// TwinCAT 3 PLC project RoboConnect
// Title: RoboConnect
// Company: RoboConnect
// Author: RoboConnect_Maintainers
// ProjectVersion: 0.1.0.1
// Description: 0.1.0.0 - Update branding 0.0.25.X Adds free taks methods 0.0.24.X Addes Manufacturer & Model to TcRobot 0.0.23.x WIP Changes pos to CartesianPos, adds GetJointPositions method 0.0.22.x WIP - adds Mode prop to interface and E_RobotModeStatus 0.0.21.0 removes task from connect 0.0.20.x modifies to newr jog approach. 0.0.19.x WIP 0.0.19.0 renames Param as causes issues in dependant libs 0.0.18.0 modifies connection and taskpool 0.0.0.17 fixes queue clear method 0.0.0.16 Updates array sizes, tcp connection and other bits 0.0.0.12 changes to TCP_Recv 0.0.0.11 adds command result tasks 0.0.010 minor change to results. 0.0.0.9 added result for tasks 0.0.0.9 added timeout for tasks 0.0.0.8 added TCP receive 0.0.0.7 removes mobject queue 0.0.0.6 adds I_CommandInvoker 0.0.0.5 I_Task extends queryable 0.0.0.4 adds logging 0.0.0.3
// ProgramVersion: 3.1.4024.0
// libraries:
//   Intecre.Utilities, * (Intecre Ltd)
//   Tc2_Standard, * (Beckhoff Automation GmbH)
//   Tc2_System, * (Beckhoff Automation GmbH)
//   Tc2_TcpIp, * (Beckhoff Automation GmbH)
// project tree:
//   CommandPattern/CommandInvoker/ I_CommandInvoker.TcIO, T_CommandInvoker.TcPOU
//   CommandPattern/CommandQueue/ E_CommandPriority.TcDUT, I_CommandQueue.TcIO, T_CommandQueue.TcPOU
//   Connection/ I_Connection.TcIO, RecvBuffer.TcDUT, T_ConnectionTCPIP.TcPOU
//   Connection/Tools/ T_TcpClientConnection.TcPOU, T_TcpRecieve.TcPOU, T_TcpSend.TcPOU
//   Helpers/ F_IsAtPositionCartesian.TcPOU, F_IsAtPositionJoint.TcPOU
//   Structs and Enums/Enum/ E_BufferMode.TcDUT, E_JogType.TcDUT
//   Structs and Enums/Struct/ ST_CartesianPoint.TcDUT, ST_Dynamics.TcDUT
//   / I_RoboConnect.TcIO, RoboConnectParams.TcGVL
//   Task/ T_BoolCommandTask_1.TcPOU (excluded from build), T_CommandTask_1.TcPOU (excluded from build), T_NumberCommandTask_1.TcPOU (excluded from build), I_CommandTask.TcIO, I_Task.TcIO, I_TaskPool.TcIO, T_TaskQueue.TcPOU
//   Project Information/ F_GetCompany.TcPOU, F_GetTitle.TcPOU, F_GetVersion.TcPOU
//   Task/ResultTasks/ I_BoolResultTask.TcIO, I_NumberResultTask.TcIO
//   Version/ Global_Version.TcGVL
// real-time tasks:
//   TASK PlcTask: cycle T#10ms, priority 22, ADS port 350
//   TASK PlcTask1: cycle T#10ms, priority 21, ADS port 351

// ---- CommandPattern/CommandQueue/E_CommandPriority.TcDUT
{attribute 'qualified_only'}
{attribute 'strict'}
{attribute 'to_string'}
TYPE E_CommandPriority :
(
	LOW := 0,
  NORMAL,
  HIGH
);
END_TYPE

// ---- Connection/RecvBuffer.TcDUT
TYPE RecvBuffer : ARRAY[1..RoboConnectParams.receiveBufferSize] OF BYTE; END_TYPE

// ---- Structs and Enums/Enum/E_BufferMode.TcDUT
{attribute 'qualified_only'}
{attribute 'strict'}
TYPE
E_BufferMode :
(
  Aborting := 0,
  Buffered := 1,
  BlendingJoint := 6,
  BlendingCartesian := 7
);
END_TYPE

// ---- Structs and Enums/Enum/E_JogType.TcDUT
{attribute 'qualified_only'}
{attribute 'strict'}
TYPE E_JogType :
(
	Joint,
  Cartesian
);
END_TYPE

// ---- Structs and Enums/Struct/ST_CartesianPoint.TcDUT
TYPE ST_CartesianPoint :
STRUCT
  x : LREAL;
  y : LREAL;
  z : LREAL;
  a : LREAL;
  b : LREAL;
  c : LREAL;
END_STRUCT
END_TYPE

// ---- Structs and Enums/Struct/ST_Dynamics.TcDUT
TYPE ST_Dynamics :
STRUCT
  Velocity : LREAL;
  Accleration : LREAL;
  Deceleration : LREAL;
END_STRUCT
END_TYPE

// ---- RoboConnectParams.TcGVL
VAR_GLOBAL CONSTANT
	receiveBufferSize : UINT := 2048;
	TimeOut : TIME := T#25S;
	MAX_TASK_SIZE : UINT := 20;
END_VAR

// ---- Version/Global_Version.TcGVL
{attribute 'TcGenerated'}
{attribute 'no-analysis'}
{attribute 'linkalways'}
// This function has been automatically generated from the project information.
VAR_GLOBAL CONSTANT
	{attribute 'const_non_replaced'}
	stLibVersion_RoboConnect : ST_LibVersion := (iMajor := 0, iMinor := 1, iBuild := 0, iRevision := 1, nFlags := 0, sVersion := '0.1.0.1');
END_VAR

// ---- CommandPattern/CommandInvoker/I_CommandInvoker.TcIO
INTERFACE I_CommandInvoker

METHOD PUBLIC CyclicLogic
END_METHOD

METHOD PUBLIC Initialise : BOOL
VAR_INPUT
  commandQueue : I_CommandQueue;
END_VAR
END_METHOD

METHOD PUBLIC Reset
END_METHOD

END_INTERFACE

// ---- CommandPattern/CommandQueue/I_CommandQueue.TcIO
INTERFACE I_CommandQueue

METHOD AddHighPriority : BOOL
VAR_INPUT
  cmd : I_Task; 
END_VAR
END_METHOD

METHOD AddLowPriority : BOOL
VAR_INPUT
  cmd : I_Task; 
END_VAR
END_METHOD

METHOD AddNormalPriority : BOOL
VAR_INPUT
  cmd : I_Task; 
END_VAR
END_METHOD

METHOD Clear
END_METHOD

PROPERTY Count : UINT
GET
END_GET
END_PROPERTY

METHOD GetNext : BOOL;
VAR_OUTPUT
	output_command : I_Task;
END_VAR
END_METHOD

END_INTERFACE

// ---- Connection/I_Connection.TcIO
INTERFACE I_Connection

METHOD Connect 
VAR_INPUT
  ip : T_IPv4Addr;
  port : UINT;
  timeout : TIME;
END_VAR
END_METHOD

METHOD Disconnect
END_METHOD

PROPERTY ErrID : UDINT
GET
END_GET
END_PROPERTY

METHOD ErrorReceive : BOOL
VAR_INPUT
END_VAR
END_METHOD

PROPERTY IsBusy : BOOL
GET
END_GET
END_PROPERTY

PROPERTY IsConnected : BOOL
GET
END_GET
END_PROPERTY

PROPERTY IsErrorConnect : Bool
GET
END_GET
END_PROPERTY

PROPERTY IsErrorReceive : Bool
GET
END_GET
END_PROPERTY

PROPERTY IsErrorSend : Bool
GET
END_GET
END_PROPERTY

METHOD Receive : BOOL // TRUE if new data recieved.
VAR_OUTPUT 
  data : ARRAY [1..RoboConnectParams.receiveBufferSize] OF BYTE;  // Contents of received buffer
  receiveLength : UDINT; // length of data received.
END_VAR
END_METHOD

METHOD Send : BOOL
VAR_INPUT
  message : T_Maxstring;
END_VAR
END_METHOD

PROPERTY PUBLIC SendDone : BOOL
GET
END_GET
END_PROPERTY

END_INTERFACE

// ---- I_RoboConnect.TcIO
INTERFACE I_RoboConnect

PROPERTY CartesianPosition : ST_CartesianPoint
GET
END_GET
END_PROPERTY

METHOD ClearError : BOOL
VAR_OUTPUT
  task : I_Task;
END_VAR
END_METHOD

METHOD Connect : BOOL
//VAR_OUTPUT
//  task : I_Task;
//END_VAR
END_METHOD

PROPERTY Connected : BOOL
GET
END_GET
END_PROPERTY

METHOD CyclicLogic
END_METHOD

METHOD Disable : BOOL
VAR_OUTPUT
  task : I_Task;
END_VAR
END_METHOD

METHOD Disconnect : BOOL
VAR_OUTPUT
  task : I_Task;
END_VAR
END_METHOD

METHOD Enable : BOOL
VAR_OUTPUT
  task : I_Task;
END_VAR
END_METHOD

PROPERTY Enabled : BOOL
GET
END_GET
END_PROPERTY

PROPERTY Error : BOOL
GET
END_GET
END_PROPERTY

PROPERTY ErrorID : LREAL
GET
END_GET
END_PROPERTY

METHOD FreeAllTasks
END_METHOD

METHOD GetAnalogOutput : BOOL
VAR_INPUT
  Index : UINT;
END_VAR
VAR_OUTPUT
  task : I_NumberResultTask;
END_VAR
END_METHOD

METHOD GetAxisCurrents : BOOL
VAR_IN_OUT
  Values : ARRAY[*] OF LREAL;
END_VAR
VAR_OUTPUT
  task : I_Task;
END_VAR
END_METHOD

METHOD GetAxisPositions : BOOL
VAR_IN_OUT
  Values : ARRAY[*] OF LREAL;
END_VAR
VAR_OUTPUT
  task : I_Task;
END_VAR
END_METHOD

METHOD GetAxisTemperatures : BOOL
VAR_IN_OUT
  Values : ARRAY[*] OF LREAL;
END_VAR
VAR_OUTPUT
  task : I_Task;
END_VAR
END_METHOD

METHOD GetDigitalOutput : BOOL
VAR_INPUT
    Index : UINT;
END_VAR
VAR_OUTPUT
  task : I_BoolResultTask;
  value 	: BOOL;
END_VAR
END_METHOD

METHOD GetJointPositions : BOOL // false if incompatible array length
VAR_IN_OUT
  joints : ARRAY[*] OF LREAL; // values overwritten with joint positions.
END_VAR
END_METHOD

METHOD GetToolAnalogOutput : BOOL
VAR_INPUT
  Index : UINT;
END_VAR
VAR_OUTPUT
  task : I_NumberResultTask;
END_VAR
END_METHOD

METHOD GetToolDigitalOutput : BOOL
VAR_INPUT
  Index : UINT;
END_VAR
VAR_OUTPUT
  task : I_BoolResultTask;
END_VAR
END_METHOD

METHOD Halt : BOOL
VAR_OUTPUT
  task : I_Task;
END_VAR
END_METHOD

METHOD IsAtCartesianPosition : BOOL
VAR_INPUT
	point	: ST_CartesianPoint;
END_VAR
END_METHOD

METHOD IsAtJointPosition : BOOL
VAR_IN_OUT
  joints : ARRAY[*] OF LREAL; // positions 1..NumberOfAxes will be used. passed array should be dimensioned accordingly
END_VAR
END_METHOD

METHOD JogAxis : BOOL // default tool and user frame
VAR_INPUT
  axisIndex : UDINT; // joint or enumerated cartesian direction/vector. See concrete type docs for enumeration of cartesian coords.
  axisDirection : BOOL; // TRUE = positive, FALSE = negative
  jogType : E_JogType; // Cartesian or Joint space
END_VAR
VAR_OUTPUT
  task : I_Task;
END_VAR
END_METHOD

METHOD JogAxisAdvanced : BOOL
VAR_INPUT
  axisIndex : UDINT; // joint or enumerated cartesian direction/vector. See concrete type docs for enumeration of cartesian coords.
  axisDirection : BOOL; // TRUE = positive, FALSE = negative
  jogType : E_JogType; // Cartesian or Joint space
  coordType : INT; // set to 0 to leave default
  user : INT; // set to 0 to leave default
  tool : INT; // set to 0 to leave default
END_VAR
VAR_OUTPUT
  task : I_Task;
END_VAR
END_METHOD

{attribute 'monitoring' : 'variable'}
PROPERTY Manufacturer : STRING
GET
END_GET
END_PROPERTY

{attribute 'monitoring' : 'variable'}
PROPERTY Model : STRING
GET
END_GET
END_PROPERTY

METHOD MoveAbs : BOOL
VAR_INPUT
  point : ST_CartesianPoint;
END_VAR
VAR_OUTPUT
  task : I_Task;
END_VAR
END_METHOD

METHOD MoveJ : BOOL
VAR_IN_OUT
  joints : ARRAY[*] OF LREAL;
END_VAR
VAR_OUTPUT
  task : I_Task;
END_VAR
END_METHOD

METHOD Reset : BOOL
VAR_OUTPUT
  task : I_Task;
END_VAR
END_METHOD

PROPERTY Running : BOOL
GET
END_GET
END_PROPERTY

METHOD SetAnalogOutput : BOOL
VAR_INPUT
  Index : UINT;
  Value : LREAL;
END_VAR
VAR_OUTPUT
  task : I_Task;
END_VAR
END_METHOD

METHOD SetAtPosDeltas : BOOL
VAR_INPUT
  atPosCartesianDeltas : ST_CartesianPoint;
END_VAR
VAR_IN_OUT
  atPosJointDeltas : ARRAY[*] OF LREAL; // positions 1..NumberOfAxes will be used. passed array should be dimensioned accordingly
END_VAR
END_METHOD

METHOD SetBufferMode : BOOL
VAR_INPUT
  BufferMode : E_BufferMode;
END_VAR
END_METHOD

METHOD SetCarteasianAcceleration : BOOL
VAR_INPUT
  Acceleration : LREAL;
END_VAR
VAR_OUTPUT
  task : I_Task;
END_VAR
END_METHOD

METHOD SetCartesianSpeed : BOOL
VAR_INPUT
  Speed : LREAL;
END_VAR
VAR_OUTPUT
  task : I_Task;
END_VAR
END_METHOD

METHOD SetDigitalOutput : BOOL
VAR_INPUT
  Index : UINT;
  Value : BOOL;
END_VAR
VAR_OUTPUT
  task : I_Task;
END_VAR
END_METHOD

METHOD SetJointAcceleration : BOOL
VAR_INPUT
  Acceleration : LREAL;
END_VAR
VAR_OUTPUT
  task : I_Task;
END_VAR
END_METHOD

METHOD SetJointSpeed : BOOL
VAR_INPUT
  Speed : LREAL;
END_VAR
VAR_OUTPUT
  task : I_Task;
END_VAR
END_METHOD

METHOD SetToolAnalogOutput : BOOL
VAR_INPUT
  Index : UINT;
  Value : LREAL;
END_VAR
VAR_OUTPUT
  task : I_Task;
END_VAR
END_METHOD

METHOD SetToolDigitalOutput : BOOL
VAR_INPUT
  Index : UINT;
  Value : BOOL;
END_VAR
VAR_OUTPUT
  task : I_Task;
END_VAR
END_METHOD

METHOD SetToolFrame : BOOL
VAR_INPUT
 Frame : ST_CartesianPoint;
END_VAR
VAR_OUTPUT
  task : I_Task;
END_VAR
END_METHOD

METHOD SetTransitionMode : BOOL
VAR_INPUT
END_VAR
END_METHOD

METHOD SetTransitionParameter : BOOL
VAR_INPUT
  CPratio : LREAL;
END_VAR
VAR_OUTPUT
	task	: I_Task;
END_VAR
END_METHOD

METHOD SetUserFrame : BOOL
VAR_INPUT
  Frame : ST_CartesianPoint;
END_VAR
VAR_OUTPUT
	task : I_Task;
END_VAR
END_METHOD

METHOD Stop : BOOL
VAR_OUTPUT
  task : I_Task;
END_VAR
END_METHOD

PROPERTY ToolPosition : ST_CartesianPoint
GET
END_GET
END_PROPERTY

END_INTERFACE

// ---- Task/I_CommandTask.TcIO
INTERFACE I_CommandTask EXTENDS I_Task

METHOD PUBLIC Initalise : BOOL
VAR_INPUT
 comPort : I_Connection;
 msg : T_Maxstring;
END_VAR
END_METHOD

END_INTERFACE

// ---- Task/I_Task.TcIO
INTERFACE I_Task EXTENDS __SYSTEM.IQueryInterface

METHOD Abort
END_METHOD

PROPERTY Available : BOOL
GET
END_GET
END_PROPERTY

PROPERTY Busy : bool
GET
END_GET
END_PROPERTY

METHOD CyclicLogic
END_METHOD

PROPERTY Done : bool
GET
END_GET
END_PROPERTY

PROPERTY Error : bool
GET
END_GET
END_PROPERTY

PROPERTY PUBLIC ErrorId : STRING
GET
END_GET
END_PROPERTY

METHOD PUBLIC Execute : BOOL
END_METHOD

METHOD PUBLIC Free
END_METHOD

PROPERTY Timeout : BOOL
GET
END_GET
END_PROPERTY

END_INTERFACE

// ---- Task/I_TaskPool.TcIO
INTERFACE I_TaskPool

METHOD PUBLIC FreeAllTasks
END_METHOD

METHOD PUBLIC GetTask : BOOL
VAR_OUTPUT
  result : I_CommandTask;
END_VAR
END_METHOD

END_INTERFACE

// ---- Task/ResultTasks/I_BoolResultTask.TcIO
INTERFACE I_BoolResultTask EXTENDS I_Task

PROPERTY Result : BOOL
GET
END_GET
END_PROPERTY

END_INTERFACE

// ---- Task/ResultTasks/I_NumberResultTask.TcIO
INTERFACE I_NumberResultTask EXTENDS I_Task

PROPERTY Result : LREAL
GET
END_GET
END_PROPERTY

END_INTERFACE

// ---- CommandPattern/CommandInvoker/T_CommandInvoker.TcPOU
FUNCTION_BLOCK T_CommandInvoker EXTENDS T_NamedBase IMPLEMENTS I_CommandInvoker
VAR
  _commandQueue : I_CommandQueue;
  currentCmd : I_Task;
  
  state, prevState : (IDLE_STATE, GET_COMMAND, PROCESSING_STATE, ERROR_STATE) := IDLE_STATE;
  initialised : BOOL;
END_VAR

METHOD PUBLIC CyclicLogic
IF NOT initialised THEN
  RETURN;
END_IF

StateMachine();
END_METHOD

PROPERTY PUBLIC Error : BOOL
GET
Error := (STATE = ERROR_STATE);
END_GET
END_PROPERTY

PROPERTY PUBLIC Idle : BOOL
GET
Idle := (STATE = IDLE_STATE);
END_GET
END_PROPERTY

METHOD PUBLIC Initialise : BOOL
VAR_INPUT
  commandQueue : I_CommandQueue;
END_VAR
IF commandQueue = 0 THEN
  LogError('command queue = 0');
  RETURN;
END_IF

LogInfo('command queue initlaised');
_commandQueue := commandQueue;

initialised := TRUE;
Initialise := TRUE;
END_METHOD

PROPERTY PUBLIC Processing : BOOL
GET
Processing := (state = PROCESSING_STATE OR STATE = GET_COMMAND);
END_GET
END_PROPERTY

METHOD PUBLIC Reset
state := IDLE_STATE;
_commandQueue.Clear();
currentCmd := 0;
END_METHOD

METHOD PRIVATE StateChanged : BOOL
IF  state = prevState THEN
  RETURN;
END_IF

prevState := state;
StateChanged := TRUE;
END_METHOD

METHOD PRIVATE StateMachine
IF currentCmd <> 0 THEN
  currentCmd.CyclicLogic();
END_IF

CASE state OF
  IDLE_STATE:
    stateChanged();

    IF _commandQueue.Count > 0 THEN
      state := GET_COMMAND;
    END_IF

  GET_COMMAND:
    StateChanged();

    IF _commandQueue.GetNext(output_command => currentCmd) THEN
      state := PROCESSING_STATE;
    END_IF

  PROCESSING_STATE:

    IF StateChanged() THEN
      
      IF currentCmd = 0 THEN
        LogError('Command invoker target task is null');
        state := ERROR_STATE;
        RETURN;

      ELSE
        currentCmd.Execute();

      END_IF
      
    ELSIF currentCmd.Done THEN
      state := IDLE_STATE;
      
    END_IF

  ERROR_STATE:
    StateChanged();

END_CASE
END_METHOD

END_FUNCTION_BLOCK

// ---- CommandPattern/CommandQueue/T_CommandQueue.TcPOU
FUNCTION_BLOCK T_CommandQueue EXTENDS T_NamedBase IMPLEMENTS I_CommandQueue
VAR
  low : T_TaskQueue;
  normal : T_TaskQueue;
  high : T_TaskQueue;
END_VAR
VAR CONSTANT
	BUFFERSIZE : UINT := 32;
END_VAR

METHOD AddHighPriority : BOOL
VAR_INPUT
  cmd : I_Task; 
END_VAR
AddHighPriority := AddWithPriority(cmd, E_CommandPriority.HIGH);
END_METHOD

METHOD AddLowPriority : BOOL
VAR_INPUT
  cmd : I_Task; 
END_VAR
AddLowPriority := AddWithPriority(cmd, E_CommandPriority.LOW);
END_METHOD

METHOD AddNormalPriority : BOOL
VAR_INPUT
  cmd : I_Task; 
END_VAR
AddNormalPriority := AddWithPriority(cmd, E_CommandPriority.NORMAL);
END_METHOD

METHOD AddWithPriority : BOOL
VAR_INPUT
  cmd : I_Task; 
  priority : E_CommandPriority;
END_VAR
VAR
  queueRef : REFERENCE TO T_TaskQueue;
END_VAR
IF cmd = 0 THEN
  LogError('Cant AddWithPriority() - cmd = 0 ');
  RETURN;
END_IF

IF Count >= BUFFERSIZE THEN
  LogError('Cant AddWithPriority() - Count >= BUFFERSIZE');
  RETURN;
END_IF

CASE priority OF
  E_CommandPriority.LOW:
    queueRef REF= low;
  E_CommandPriority.NORMAL:
    queueRef REF= normal;
  E_CommandPriority.HIGH:
    queueRef REF= high;
ELSE
  LogError(CONCAT('Unknown priority for command: ', TO_STRING(priority)));
  RETURN;

END_CASE

AddWithPriority := queueRef.Enqueue(cmd);

LogInfo(CONCAT(TO_STRING(priority),' priority command added to queue'));
END_METHOD

METHOD Clear
low.Clear();
normal.Clear();
high.Clear();

logInfo('Command queue cleared');
END_METHOD

PROPERTY Count : UINT
GET
//Combine all three queues and return the result
Count := Dint_to_Uint(high.Count + normal.Count + low.Count);
END_GET
END_PROPERTY

METHOD GetNext : BOOL
VAR_OUTPUT
	output_command : I_Task;
END_VAR
IF high.Count > 0 THEN
  IF high.TryDequeue(result => output_command) THEN
    LogInfo('High priority item dequeued');
    GetNext := TRUE;
    RETURN;

  ELSE
    GetNext := FALSE;
    RETURN;

  END_IF
ELSIF high.Count = 0 AND normal.Count > 0 THEN

  IF normal.TryDequeue(result => output_command) THEN
    LogInfo('Normal priority item dequeued');
    GetNext := TRUE;
    RETURN;

  ELSE
    GetNext := FALSE;
    RETURN;

  END_IF

ELSIF high.Count = 0 AND normal.Count = 0 AND low.Count > 0 THEN
  IF low.TryDequeue(result => output_command) THEN
    LogInfo('Low priority item dequeued');
    GetNext := TRUE;
    RETURN;

  ELSE
    GetNext := FALSE;
    RETURN;

  END_IF
END_IF
END_METHOD

END_FUNCTION_BLOCK

// ---- Task/T_TaskQueue.TcPOU
FUNCTION_BLOCK T_TaskQueue EXTENDS T_NamedBase
VAR
  _items : ARRAY[1..QUEUE_SIZE] OF I_Task;
  _count : UINT := 0;
END_VAR
VAR CONSTANT
  QUEUE_SIZE : UINT := 10;
END_VAR

METHOD PUBLIC Clear 
VAR
	index : UINT;
END_VAR
FOR index := 1 TO _count DO
  _items[index].Abort();
END_FOR

_count := 0;
MEMSET(ADR(_items), 0, SIZEOF(_items));
END_METHOD

METHOD PUBLIC Contains : BOOL
VAR_INPUT
	Target : I_Task;
END_VAR
VAR
	i : UINT;
END_VAR
IF Target = 0 THEN
	LogError('Input is null');
	RETURN;
END_IF

FOR i := 1 TO _count DO 
	IF _items[i] = 0 THEN
		LogError('Attempted to check a null reference');
		CONTINUE;
	END_IF	

	IF target = _items[i] THEN
		Contains := TRUE;
		RETURN;
	END_IF
END_FOR

Contains := FALSE;
END_METHOD

PROPERTY Count : UINT
GET
Count := _count;
END_GET
END_PROPERTY

METHOD PUBLIC Enqueue : BOOL
VAR_INPUT
    newTask : I_Task;
END_VAR
IF _count >= QUEUE_SIZE THEN
    RETURN;

END_IF

_items[_count + 1] := newTask;
_count := _count + 1;

Enqueue := TRUE;
END_METHOD

METHOD PUBLIC TryDequeue : BOOL
VAR_OUTPUT
    result : I_Task;
END_VAR
VAR
    target : I_Task;
END_VAR
IF _count < 1 THEN
    RETURN;
END_IF

target := _items[1];
_count := _count - 1;

MEMMOVE(ADR(_items[1]), ADR(_items[2]), SIZEOF(_items) - SIZEOF(_items[1]));

result := target;
TryDequeue := TRUE;
END_METHOD

END_FUNCTION_BLOCK

// ---- Connection/Tools/T_TcpClientConnection.TcPOU
FUNCTION_BLOCK T_TcpClientConnection
VAR
    connection : FB_ClientServerConnection;
	_log : T_NamedBase;
END_VAR

METHOD PUBLIC Connect
VAR_INPUT
  ip : T_IPv4Addr;
  port : UINT;
  timeout : TIME;
END_VAR
connection.sRemoteHost := ip;
connection.nRemotePort := port;
connection.tReconnect := timeout;
connection.nMode := CONNECT_MODE_ENABLEDBG;
connection.bEnable := TRUE;
END_METHOD

METHOD PUBLIC CyclicLogic
VAR_INST
	TON_ConnectTimer : TON;
END_VAR
connection();

TON_ConnectTimer(
	IN:= connection.bEnable AND NOT IsConnected,
	PT:= connection.tReconnect,
	Q=> ,
	ET=> );

IF TON_ConnectTimer.Q THEN
	connection.bEnable := FALSE;
	_log.LogError('Connection time out');
END_IF
END_METHOD

METHOD PUBLIC Disconnect
connection.bEnable := FALSE;
_log.LogInfo('Disconnected');
END_METHOD

PROPERTY ErrID : UDINT
GET
ErrID := connection.nErrId;
END_GET
END_PROPERTY

PROPERTY PUBLIC IsBusy : BOOL
GET
IsBusy := connection.bBusy;
END_GET
END_PROPERTY

PROPERTY PUBLIC IsConnected : BOOL
GET
IsConnected := (connection.eState = E_SocketConnectionState.eSOCKET_CONNECTED);
END_GET
END_PROPERTY

PROPERTY PUBLIC IsError : BOOL
GET
IsError := connection.bError;
END_GET
END_PROPERTY

PROPERTY PUBLIC Socket : REFERENCE TO T_HSOCKET
GET
Socket REF= connection.hSocket;
END_GET
END_PROPERTY

END_FUNCTION_BLOCK

// ---- Connection/Tools/T_TcpRecieve.TcPOU
FUNCTION_BLOCK T_TcpRecieve
VAR
  receiver : FB_SocketReceive; //
  _socket : REFERENCE TO T_HSOCKET; // TCP-IP socket
  _log : T_NamedBase; //
  receiveBuffer : RecvBuffer; // Contents of received buffer
  receiveLength : UDINT; // Length of received string
  trigNotBusy : F_TRIG;
  execute : BOOL;
END_VAR

// If no open socket, return
IF NOT HasSocket THEN
  RETURN;
END_IF

receiver(
	sSrvNetId:= , 
	hSocket:= _socket, 
	cbLen:= SIZEOF(receiveBuffer), 
	pDest:= ADR(receiveBuffer), 
	bExecute:= , 
	tTimeout:= TimeOut, 
	bBusy=> , 
	bError=> , 
	nErrId=> , 
	nRecBytes=> receiveLength);
 
IF NOT execute THEN
  receiver.bExecute := FALSE;
  RETURN;
END_IF

receiver.bExecute S= NOT receiver.bExecute;

// Receiver runs as soon as socket is connected
// When bBusy goes low, check for new message
trigNotBusy(CLK:= receiver.bBusy, Q=> );

receiver.bExecute R= trigNotBusy.Q;

METHOD PUBLIC CyclicLogic
THIS^();
END_METHOD

PROPERTY ErrID : UDINT
GET
ErrID := receiver.nErrId;
END_GET
END_PROPERTY

PROPERTY INTERNAL HasSocket : BOOL
GET
HasSocket := __ISVALIDREF(_socket);
END_GET
END_PROPERTY

PROPERTY PUBLIC IsBusy : BOOL
GET
IsBusy := receiver.bBusy;
END_GET
END_PROPERTY

PROPERTY PUBLIC IsError : BOOL
GET
IsError := receiver.bError;
END_GET
END_PROPERTY

METHOD INTERNAL SetSocket : BOOL
VAR_IN_OUT
  socket : T_HSOCKET;
END_VAR
_socket REF= socket;
_log.LogDebug('SetSocket := TRUE');
SetSocket := TRUE;
END_METHOD

METHOD Start // starts receiving
execute := TRUE;
END_METHOD

METHOD Stop // stops receiving. Must be called if socket dies.
execute := FALSE;
END_METHOD

METHOD PUBLIC TryGetBuffer : BOOL
VAR_IN_OUT
  result : RecvBuffer;
END_VAR
VAR_OUTPUT
  receiveLength : UDINT;
END_VAR
IF NOT HasSocket THEN
  _log.LogError('Cannot Receive as NOT HasSocket');
  RETURN;

END_IF

TryGetBuffer := THIS^.receiveLength > 0;

IF NOT TryGetBuffer THEN
  RETURN;
  
END_IF

result := receiveBuffer; // copy by val into referenced buffer
receiveLength := THIS^.receiveLength;

THIS^.receiveLength := 0;
MEMSET(ADR(receiveBuffer), 0, SIZEOF(receiveBuffer));
END_METHOD

END_FUNCTION_BLOCK

// ---- Connection/Tools/T_TcpSend.TcPOU
FUNCTION_BLOCK T_TcpSend
VAR
	sender : FB_SocketSend;
	_socket : REFERENCE TO T_HSOCKET;	// TCP-IP socket
	_log : T_NamedBase;
	_message : T_MAXSTRING;				// Message to send
END_VAR

METHOD PUBLIC CyclicLogic
IF NOT __ISVALIDREF(_socket) THEN
  RETURN;
END_IF

sender(
	sSrvNetId:= , 
	hSocket:= _socket, 
	cbLen:= TO_UDINT(LEN(_message)), 
	pSrc:= ADR(_message), 
	bExecute:= , 
	tTimeout:= TimeOut, 
	bBusy=> , 
	bError=> , 
	nErrId=> );

IF NOT sender.bBusy THEN
  sender.bExecute := FALSE;
END_IF

IF sender.bError THEN
	_log.LogError('Send Error');
END_IF
END_METHOD

PROPERTY ErrID : UDINT
GET
ErrID := sender.nErrId;
END_GET
END_PROPERTY

PROPERTY INTERNAL HasSocket : BOOL
GET
HasSocket := __ISVALIDREF(_socket);
END_GET
END_PROPERTY

PROPERTY PUBLIC IsBusy : BOOL
GET
IsBusy := sender.bBusy;
END_GET
END_PROPERTY

PROPERTY PUBLIC IsError : BOOL
GET
IsError := sender.bError;
END_GET
END_PROPERTY

METHOD PUBLIC Send : BOOL;
VAR_INPUT
  message : T_MAXSTRING; 
END_VAR
IF NOT HasSocket THEN
  _log.LogError('Cannot Send as NOT HasSocket');
  RETURN;

END_IF

_message := message;
sender.bExecute := TRUE;
Send := TRUE;
END_METHOD

METHOD INTERNAL SetSocket : BOOL
VAR_IN_OUT
  socket : T_HSOCKET;
END_VAR
_socket REF= socket;
_log.LogDebug('SetSocket := TRUE');
SetSocket := TRUE;
END_METHOD

END_FUNCTION_BLOCK

// ---- Connection/T_ConnectionTCPIP.TcPOU
FUNCTION_BLOCK T_ConnectionTCPIP EXTENDS T_NamedBase IMPLEMENTS I_Connection
VAR
	connection : T_TcpClientConnection;
	sender : T_TcpSend;
	receiver : T_TcpRecieve;
	init : BOOL;
	state : (IDLE, WORKING);
  
  IsConnectedTrigger : R_TRIG;
  IsNotConnectedTrigger : F_TRIG;
END_VAR

METHOD Connect 
VAR_INPUT
  ip : T_IPv4Addr;
  port : UINT;
  timeout : TIME;
END_VAR
connection.Connect(ip, port, timeout);
LogInfo('Connecting');
END_METHOD

METHOD PUBLIC CyclicLogic
VAR_INST
  trigConnected : R_TRIG;
  isNotConnectedTrigger : F_TRIG;
  trigErrReceive : R_TRIG;
END_VAR
IF NOT init THEN
	init := TRUE;
END_IF

connection.CyclicLogic();
trigConnected(CLK := connection.IsConnected);

IF trigConnected.Q THEN
	sender.SetSocket(connection.Socket);
	receiver.SetSocket(connection.Socket);
  receiver.Start();
	LogDebug('Connected - setting socket on sender and receiver.');
END_IF

isNotConnectedTrigger(CLK := connection.IsConnected);
IF isNotConnectedTrigger.Q THEN
  receiver.Stop();
END_IF

IF NOT connection.IsConnected THEN
 	RETURN;
END_IF

sender.CyclicLogic();
receiver.CyclicLogic();

// If error detected on receive, need to try disconnecting and reconnecting
trigErrReceive(CLK:= IsErrorReceive, Q=> );
IF trigErrReceive.Q THEN
	ErrorReceive();
END_IF
END_METHOD

METHOD Disconnect
connection.Disconnect();
LogInfo('Disconnecting');
END_METHOD

PROPERTY ErrID : UDINT
GET
IF IsErrorConnect THEN
	ErrID := connection.ErrID;
ELSIF IsErrorSend THEN
	ErrID := sender.ErrID;
ELSIF IsErrorReceive THEN
	ErrID := receiver.ErrID;
END_IF
END_GET
END_PROPERTY

METHOD ErrorReceive : BOOL
LogError('Receive Error');
Disconnect();
END_METHOD

PROPERTY IsBusy : BOOL
GET
IsBusy := connection.IsBusy OR sender.IsBusy OR receiver.IsBusy;
END_GET
END_PROPERTY

PROPERTY IsConnected : BOOL
GET
IsConnected := connection.IsConnected;
END_GET
END_PROPERTY

PROPERTY IsErrorConnect : Bool
GET
IsErrorConnect := connection.IsError;
END_GET
END_PROPERTY

PROPERTY IsErrorReceive : BOOL
GET
IsErrorReceive := receiver.IsError;
END_GET
END_PROPERTY

PROPERTY IsErrorSend : BOOL
GET
IsErrorSend := sender.IsError;
END_GET
END_PROPERTY

METHOD Receive : BOOL // TRUE if new data recieved.
VAR_OUTPUT 
  data : ARRAY [1..RoboConnectParams.receiveBufferSize] OF BYTE;  // Contents of received buffer
  receiveLength : UDINT; // length of data received.
END_VAR
IF NOT connection.IsConnected THEN
  LogWarning('Cannot receive message, NOT connected');
  RETURN;
END_IF

Receive :=
  receiver.TryGetBuffer(
    result := data,
    receiveLength => receiveLength
  );
END_METHOD

METHOD Send : BOOL
VAR_INPUT
  message : T_Maxstring;
END_VAR
IF NOT connection.IsConnected THEN
  LogWarning('Cannot send message, not connected');
  RETURN;
END_IF

LogInfo(CONCAT('Sending message : ', message));
sender.Send(message);
Send := TRUE;
END_METHOD

PROPERTY PUBLIC SendDone : BOOL
GET
SendDone := NOT sender.IsBusy;
END_GET
END_PROPERTY

END_FUNCTION_BLOCK

// ---- Helpers/F_IsAtPositionCartesian.TcPOU
FUNCTION F_IsAtPositionCartesian : BOOL
VAR_INPUT
  actual : ST_CartesianPoint;
  target : ST_CartesianPoint;
  delta : ST_CartesianPoint;
END_VAR

F_IsAtPositionCartesian :=
  (ABS(actual.x - target.x) < delta.x)
    AND (ABS(actual.x - target.x) < delta.x)
    AND (ABS(actual.y - target.y) < delta.y)
    AND (ABS(actual.z - target.z) < delta.z)
    AND (ABS(actual.a - target.a) < delta.a)
    AND (ABS(actual.b - target.b) < delta.b)
    AND (ABS(actual.c - target.c) < delta.c);

END_FUNCTION

// ---- Helpers/F_IsAtPositionJoint.TcPOU
FUNCTION F_IsAtPositionJoint : BOOL
VAR_IN_OUT
  actual : ARRAY[*] OF LREAL;
  target : ARRAY[*] OF LREAL;
  delta  : ARRAY[*] OF LREAL;
END_VAR
VAR
  actLower, actUpper : DINT;
  ind : DINT;
END_VAR

actLower := LOWER_BOUND(actual, 1);
actUpper := UPPER_BOUND(actual, 1); 

IF actLower > LOWER_BOUND(target,1) OR actLower > LOWER_BOUND(delta, 1) THEN
  F_LogWarning('actLower > LOWER_BOUND(target,1) OR actLower > LOWER_BOUND(delta, 1)');
  RETURN;
  
END_IF

IF actUpper > UPPER_BOUND(target,1) OR actLower > UPPER_BOUND(delta, 1) THEN
  F_LogWarning('actUpper > UPPER_BOUND(target,1) OR actLower > UPPER_BOUND(delta, 1)');
  RETURN;
  
END_IF

FOR ind := actLower TO actUpper DO
  F_IsAtPositionJoint := ABS(actual[ind] - target[ind]) < delta[ind];
  
  IF NOT F_IsAtPositionJoint THEN
    // any failure means not in position.
    RETURN;
    
	END_IF
  
END_FOR

END_FUNCTION

// ---- Task/T_BoolCommandTask_1.TcPOU
FUNCTION_BLOCK T_BoolCommandTask_1 EXTENDS T_MockCommandTask IMPLEMENTS I_BoolResultTask
VAR
  _result : BOOL;
END_VAR

PROPERTY Result : BOOL
GET
Result := _result;
END_GET
END_PROPERTY

METHOD PUBLIC SetResultValue
VAR_INPUT
  value : BOOL;
END_VAR
_result := value;
END_METHOD

END_FUNCTION_BLOCK

// ---- Task/T_CommandTask_1.TcPOU
FUNCTION_BLOCK T_CommandTask_1 EXTENDS T_NamedBase IMPLEMENTS I_CommandTask
VAR_INPUT
  _busy : BOOL := FALSE;
  _error : BOOL := FALSE;
  _done : BOOL := FALSE;
  _timeout : BOOL := FALSE;
  _available : BOOL := TRUE;
END_VAR
VAR

  _errorId : STRING;
  _msg : T_Maxstring;
  timeoutTimer : TON := (PT := TASK_TIMEOUT);

  state, prevState : (UNINITLIASED,
    INITALISED,
    EXECUTING,
    DONE_STATE,
    ERROR_STATE);

END_VAR
VAR CONSTANT
  TASK_TIMEOUT : TIME := RoboConnectParams.TimeOut;
END_VAR

METHOD Abort
END_METHOD

PROPERTY Available : BOOL
GET
Available := _available;
END_GET
END_PROPERTY

PROPERTY Busy : BOOL
GET
Busy := _Busy;
END_GET
END_PROPERTY

METHOD PUBLIC CyclicLogic



CASE state OF
  UNINITLIASED:
    StateChanged();

  INITALISED:
    IF StateChanged() THEN
      logInfo('task initlaised');
    END_IF

  EXECUTING:
    IF StateChanged() THEN
      LogInfo('task executing');
      _busy := TRUE;
      timeoutTimer.IN := TRUE;
      
      IF NOT _comPort.Send(_msg) THEN
        state := ERROR_STATE;
        RETURN;
			END_IF
      
    END_IF
    
    IF timeoutTimer.Q THEN
      state := ERROR_STATE;
      LogError('Command timed out');
		END_IF

    IF _comPort.SendDone THEN
      state := DONE_STATE;
    END_IF

  DONE_STATE:
    IF StateChanged() THEN
      LogInfo('task done');
      _busy := FALSE;
      _done := TRUE;
      timeoutTimer.IN := FALSE;
    END_IF

  ERROR_STATE:
    IF StateChanged() THEN
      LogError('task error');
      _error := TRUE;
      _busy := FALSE;
      _done := FALSE;
    END_IF

END_CASE

timeoutTimer();
END_METHOD

PROPERTY Done : BOOL
GET
Done := _Done;
END_GET
END_PROPERTY

PROPERTY Error : BOOL
GET
Error := _Error;
END_GET
END_PROPERTY

PROPERTY PUBLIC ErrorId : string
GET
ErrorId := _errorId;
END_GET
END_PROPERTY

METHOD PUBLIC Execute : BOOL
IF state <> INITALISED THEN
  RETURN;
END_IF

state := EXECUTING;
EXECUTE := TRUE;
END_METHOD

METHOD PUBLIC Free
_Busy := FALSE;
_Error := FALSE;
_Done := FALSE;
 _timeout := FALSE;
 _available := TRUE;
  
_comPort := 0;
_msg := '';
END_METHOD

METHOD PUBLIC Initalise : BOOL
VAR_INPUT
 msg : T_Maxstring;
END_VAR
_done := FALSE;
_msg := msg;
state := INITALISED;
_available := FALSE;
Initalise := TRUE;
END_METHOD

METHOD PRIVATE StateChanged : BOOL
IF  state = prevState THEN
  RETURN;
END_IF

prevState := state;
StateChanged := TRUE;
END_METHOD

PROPERTY Timeout : BOOL
GET
Timeout := _timeout;
END_GET
END_PROPERTY

END_FUNCTION_BLOCK

// ---- Task/T_NumberCommandTask_1.TcPOU
FUNCTION_BLOCK T_NumberCommandTask_1 EXTENDS T_MockCommandTask IMPLEMENTS I_NumberResultTask
VAR
  _result : LREAL;
END_VAR

PROPERTY Result : LREAL
GET
Result := _result;
END_GET
END_PROPERTY

METHOD PUBLIC SetResultValue
VAR_INPUT
  value : LREAL;
END_VAR
_result := value;
END_METHOD

END_FUNCTION_BLOCK

// ---- Project Information/F_GetCompany.TcPOU
// This function has been automatically generated from the project information.
{attribute 'signature_flag' := '1073741824'}
{attribute 'TcGenerated'}
{attribute 'no-analysis'}
FUNCTION F_GetCompany : WSTRING
VAR_INPUT
	
END_VAR

F_GetCompany := "RoboConnect";

END_FUNCTION

// ---- Project Information/F_GetTitle.TcPOU
// This function has been automatically generated from the project information.
{attribute 'signature_flag' := '1073741824'}
{attribute 'TcGenerated'}
{attribute 'no-analysis'}
FUNCTION F_GetTitle : WSTRING
VAR_INPUT
	
END_VAR

F_GetTitle := "RoboConnect";

END_FUNCTION

// ---- Project Information/F_GetVersion.TcPOU
// This function has been automatically generated from the project information.
{attribute 'signature_flag' := '1073741824'}
{attribute 'TcGenerated'}
{attribute 'no-analysis'}
FUNCTION F_GetVersion : ST_LibVersion
VAR_INPUT
	
END_VAR

F_GetVersion.iMajor := 0;
F_GetVersion.iMinor := 1;
F_GetVersion.iBuild := 0;
F_GetVersion.iRevision := 1;
F_GetVersion.sVersion := '0.1.0.1';
F_GetVersion.nFlags := 0;

END_FUNCTION
